TYPE ST_LinCoord_XY :
STRUCT
	x	: REAL;	// [mm]
	y	: REAL;	// [mm]
END_STRUCT
END_TYPE

(* stored: Version 1.1.0.1, ProductVersion 3.1.4026.18
   DUT ST_LinCoord_XY: Id {7006fac1-d820-4c19-b5cb-80184e958f57} *)
